// TIA Portal V20 export
TYPE "typeSequenceControlNodeHomeCheck"
// stored: Namespace Unit1.Em13
   STRUCT
      partNoDetect { ExternalWritable := 'False'} : Bool;
      partDetect { ExternalWritable := 'False'} : Bool;
   END_STRUCT;
END_TYPE
